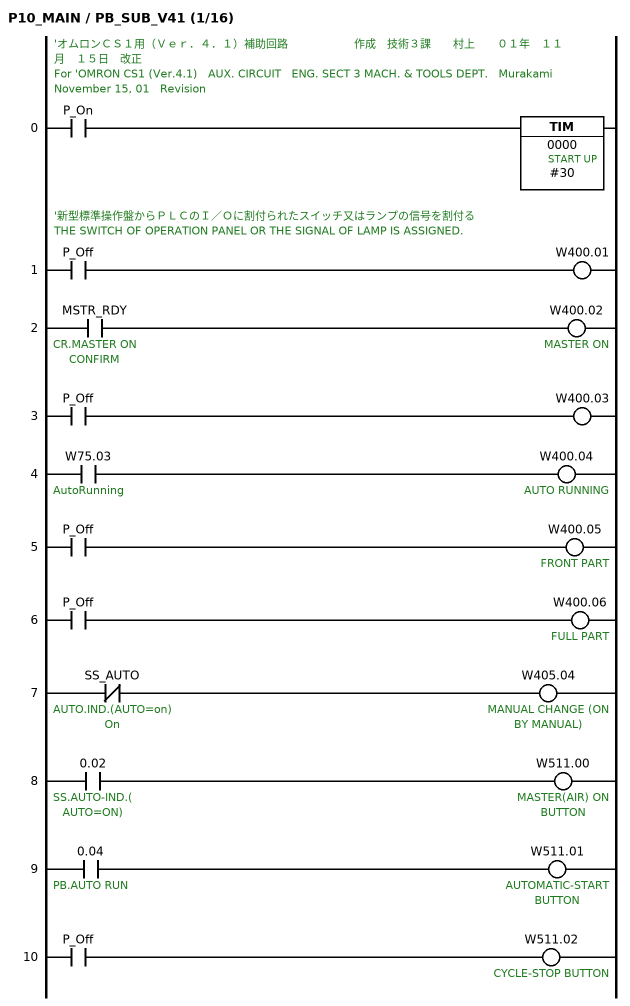
; [picture p72: P10_MAIN / PB_SUB_V41, rungs 0-10]
; rung 0: 'オムロンＣＳ１用（Ｖｅｒ．４．１）補助回路　　　　　　作成　技術３課　　村上　　０１年　１１月　１５日　改正 / For 'OMRON CS1 (Ver.4.1)   AUX. CIRCUIT   ENG. SECT 3 MACH. & TOOLS DEPT.   Murakami   November 15, 01   Revision
LD P_On
TIM 0000 #30  ; START UP
; rung 1: '新型標準操作盤からＰＬＣのＩ／Ｏに割付られたスイッチ又はランプの信号を割付る / THE SWITCH OF OPERATION PANEL OR THE SIGNAL OF LAMP IS ASSIGNED.
LD P_Off
OUT W400.01
; rung 2
LD MSTR_RDY  ; CR.MASTER ON CONFIRM
OUT W400.02  ; MASTER ON
; rung 3
LD P_Off
OUT W400.03
; rung 4
LD W75.03  ; AutoRunning
OUT W400.04  ; AUTO RUNNING
; rung 5
LD P_Off
OUT W400.05  ; FRONT PART
; rung 6
LD P_Off
OUT W400.06  ; FULL PART
; rung 7
LDNOT SS_AUTO  ; AUTO.IND.(AUTO=on) On
OUT W405.04  ; MANUAL CHANGE (ON BY MANUAL)
; rung 8
LD 0.02  ; SS.AUTO-IND.(AUTO=ON)
OUT W511.00  ; MASTER(AIR) ON BUTTON
; rung 9
LD 0.04  ; PB.AUTO RUN
OUT W511.01  ; AUTOMATIC-START BUTTON
; rung 10
LD P_Off
OUT W511.02  ; CYCLE-STOP BUTTON

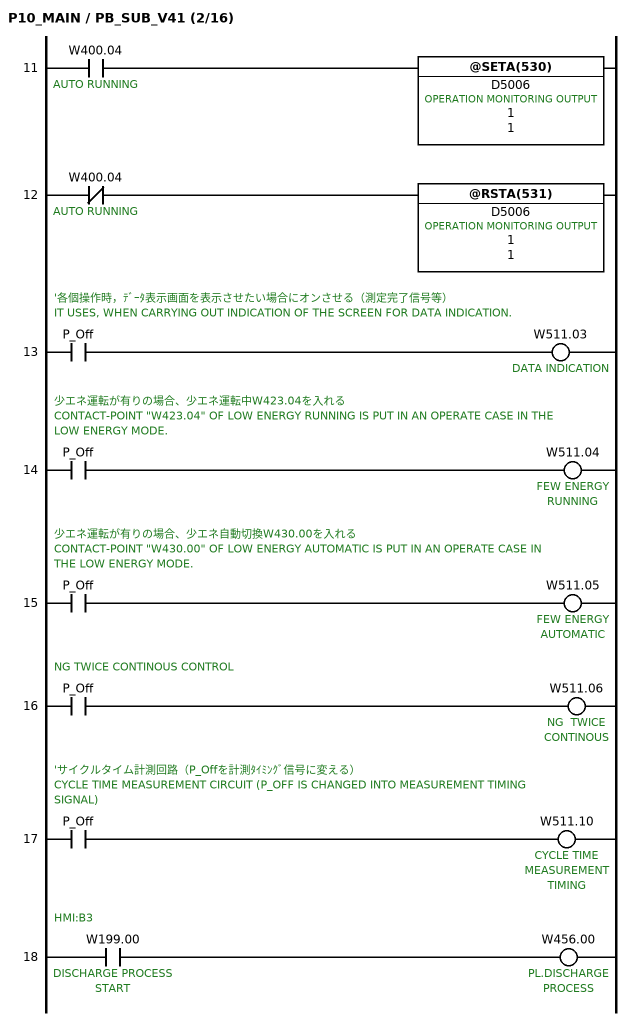
; rung 11
LD W400.04  ; AUTO RUNNING
@SETA(530) D5006 1 1  ; OPERATION MONITORING OUTPUT
; rung 12
LDNOT W400.04  ; AUTO RUNNING
@RSTA(531) D5006 1 1  ; OPERATION MONITORING OUTPUT
; rung 13: '各個操作時，ﾃﾞｰﾀ表示画面を表示させたい場合にオンさせる（測定完了信号等） / IT USES, WHEN CARRYING OUT INDICATION OF THE SCREEN FOR DATA INDICATION.
LD P_Off
OUT W511.03  ; DATA INDICATION
; rung 14: 少エネ運転が有りの場合、少エネ運転中W423.04を入れる / CONTACT-POINT "W423.04" OF LOW ENERGY RUNNING IS PUT IN AN OPERATE CASE IN THE LOW ENERGY MODE.
LD P_Off
OUT W511.04  ; FEW ENERGY RUNNING
; rung 15: 少エネ運転が有りの場合、少エネ自動切換W430.00を入れる / CONTACT-POINT "W430.00" OF LOW ENERGY AUTOMATIC IS PUT IN AN OPERATE CASE IN THE LOW ENERGY MODE.
LD P_Off
OUT W511.05  ; FEW ENERGY AUTOMATIC
; rung 16: NG TWICE CONTINOUS CONTROL
LD P_Off
OUT W511.06  ; NG  TWICE CONTINOUS
; rung 17: 'サイクルタイム計測回路（P_Offを計測ﾀｲﾐﾝｸﾞ信号に変える） / CYCLE TIME MEASUREMENT CIRCUIT (P_OFF IS CHANGED INTO MEASUREMENT TIMING SIGNAL)
LD P_Off
OUT W511.10  ; CYCLE TIME MEASUREMENT TIMING
; rung 18: HMI:B3
LD W199.00  ; DISCHARGE PROCESS START
OUT W456.00  ; PL.DISCHARGE PROCESS

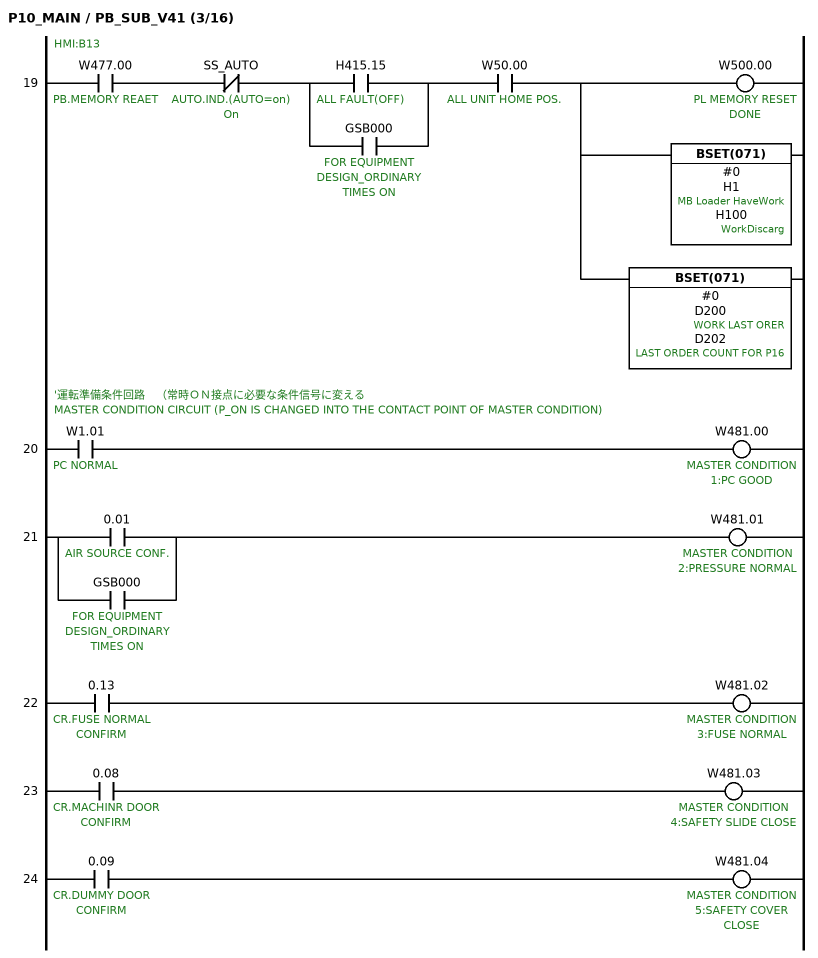
; rung 19: HMI:B13
LD W477.00  ; PB.MEMORY REAET
ANDNOT SS_AUTO  ; AUTO.IND.(AUTO=on) On
LD H415.15  ; ALL FAULT(OFF)
OR GSB000  ; FOR EQUIPMENT DESIGN_ORDINARY TIMES ON
ANDLD
AND W50.00  ; ALL UNIT HOME POS.
OUT W500.00  ; PL MEMORY RESET DONE
BSET(071) #0 H1 H100  ; MB Loader HaveWork, WorkDiscarg
BSET(071) #0 D200 D202  ; WORK LAST ORER, LAST ORDER COUNT FOR P16
; rung 20: '運転準備条件回路　（常時ＯＮ接点に必要な条件信号に変える / MASTER CONDITION CIRCUIT (P_ON IS CHANGED INTO THE CONTACT POINT OF MASTER CONDITION)
LD W1.01  ; PC NORMAL
OUT W481.00  ; MASTER CONDITION 1:PC GOOD
; rung 21
LD 0.01  ; AIR SOURCE CONF.
OR GSB000  ; FOR EQUIPMENT DESIGN_ORDINARY TIMES ON
OUT W481.01  ; MASTER CONDITION 2:PRESSURE NORMAL
; rung 22
LD 0.13  ; CR.FUSE NORMAL CONFIRM
OUT W481.02  ; MASTER CONDITION 3:FUSE NORMAL
; rung 23
LD 0.08  ; CR.MACHINR DOOR CONFIRM
OUT W481.03  ; MASTER CONDITION 4:SAFETY SLIDE CLOSE
; rung 24
LD 0.09  ; CR.DUMMY DOOR CONFIRM
OUT W481.04  ; MASTER CONDITION 5:SAFETY COVER CLOSE

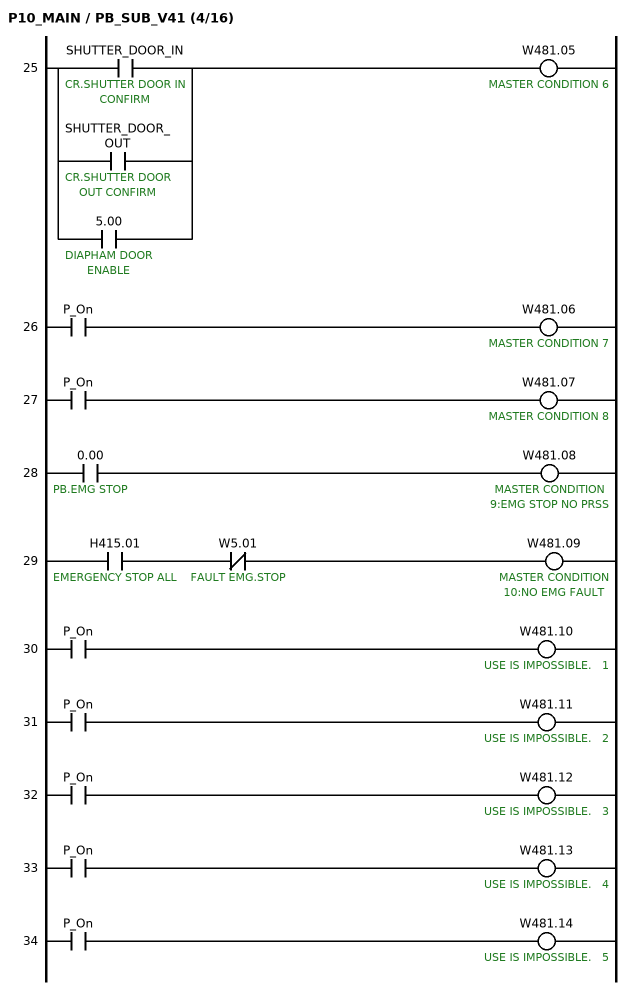
; rung 25
LD SHUTTER_DOOR_IN  ; CR.SHUTTER DOOR IN CONFIRM
OR SHUTTER_DOOR_OUT  ; CR.SHUTTER DOOR OUT CONFIRM
OR 5.00  ; DIAPHAM DOOR ENABLE
OUT W481.05  ; MASTER CONDITION 6
; rung 26
LD P_On
OUT W481.06  ; MASTER CONDITION 7
; rung 27
LD P_On
OUT W481.07  ; MASTER CONDITION 8
; rung 28
LD 0.00  ; PB.EMG STOP
OUT W481.08  ; MASTER CONDITION 9:EMG STOP NO PRSS
; rung 29
LD H415.01  ; EMERGENCY STOP ALL
ANDNOT W5.01  ; FAULT EMG.STOP
OUT W481.09  ; MASTER CONDITION 10:NO EMG FAULT
; rung 30
LD P_On
OUT W481.10  ; USE IS IMPOSSIBLE.   1
; rung 31
LD P_On
OUT W481.11  ; USE IS IMPOSSIBLE.   2
; rung 32
LD P_On
OUT W481.12  ; USE IS IMPOSSIBLE.   3
; rung 33
LD P_On
OUT W481.13  ; USE IS IMPOSSIBLE.   4
; rung 34
LD P_On
OUT W481.14  ; USE IS IMPOSSIBLE.   5

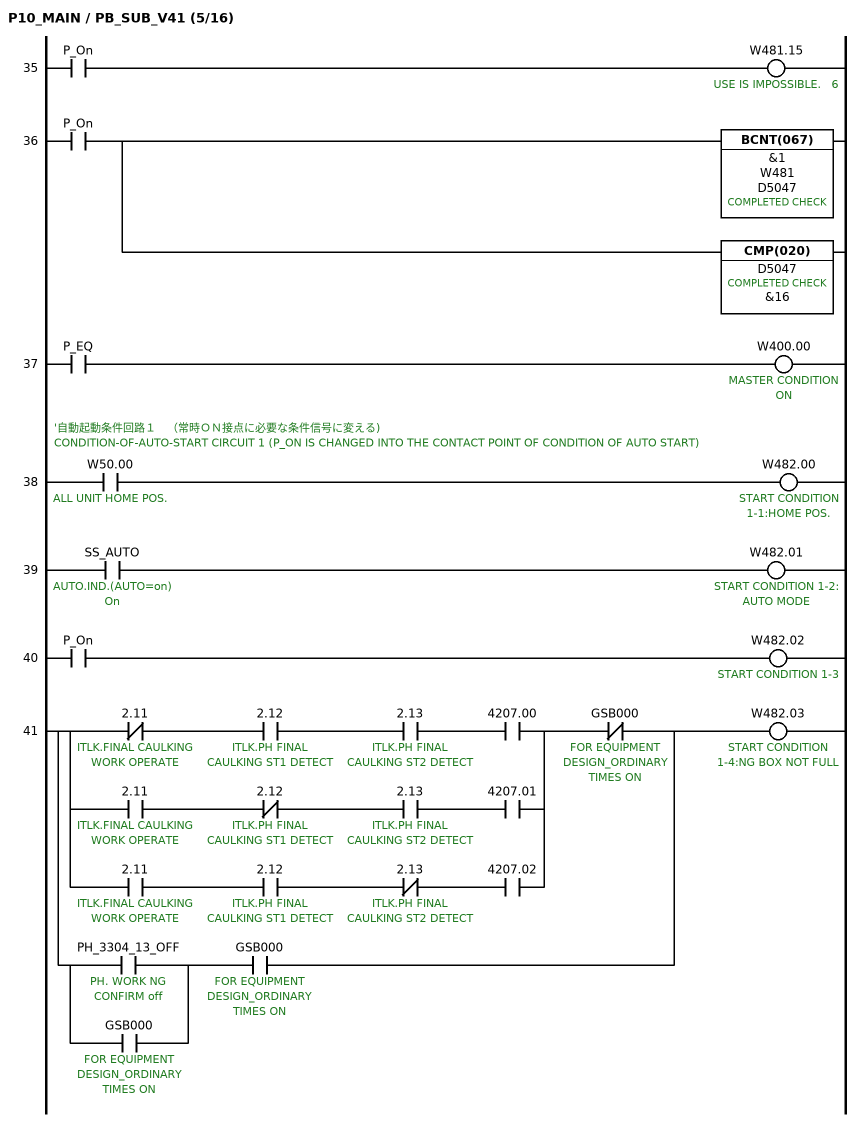
; rung 35
LD P_On
OUT W481.15  ; USE IS IMPOSSIBLE.   6
; rung 36
LD P_On
BCNT(067) &1 W481 D5047  ; COMPLETED CHECK
CMP(020) D5047 &16  ; COMPLETED CHECK
; rung 37
LD P_EQ
OUT W400.00  ; MASTER CONDITION ON
; rung 38: '自動起動条件回路１　（常時ＯＮ接点に必要な条件信号に変える) / CONDITION-OF-AUTO-START CIRCUIT 1 (P_ON IS CHANGED INTO THE CONTACT POINT OF CONDITION OF AUTO START)
LD W50.00  ; ALL UNIT HOME POS.
OUT W482.00  ; START CONDITION 1-1:HOME POS.
; rung 39
LD SS_AUTO  ; AUTO.IND.(AUTO=on) On
OUT W482.01  ; START CONDITION 1-2: AUTO MODE
; rung 40
LD P_On
OUT W482.02  ; START CONDITION 1-3
; rung 41
LDNOT 2.11  ; ITLK.FINAL CAULKING WORK OPERATE
AND 2.12  ; ITLK.PH FINAL CAULKING ST1 DETECT
AND 2.13  ; ITLK.PH FINAL CAULKING ST2 DETECT
AND 4207.00
LD 2.11  ; ITLK.FINAL CAULKING WORK OPERATE
ANDNOT 2.12  ; ITLK.PH FINAL CAULKING ST1 DETECT
AND 2.13  ; ITLK.PH FINAL CAULKING ST2 DETECT
AND 4207.01
ORLD
LD 2.11  ; ITLK.FINAL CAULKING WORK OPERATE
AND 2.12  ; ITLK.PH FINAL CAULKING ST1 DETECT
ANDNOT 2.13  ; ITLK.PH FINAL CAULKING ST2 DETECT
AND 4207.02
ORLD
ANDNOT GSB000  ; FOR EQUIPMENT DESIGN_ORDINARY TIMES ON
LD PH_3304_13_OFF  ; PH. WORK NG CONFIRM off
OR GSB000  ; FOR EQUIPMENT DESIGN_ORDINARY TIMES ON
AND GSB000  ; FOR EQUIPMENT DESIGN_ORDINARY TIMES ON
ORLD
OUT W482.03  ; START CONDITION 1-4:NG BOX NOT FULL

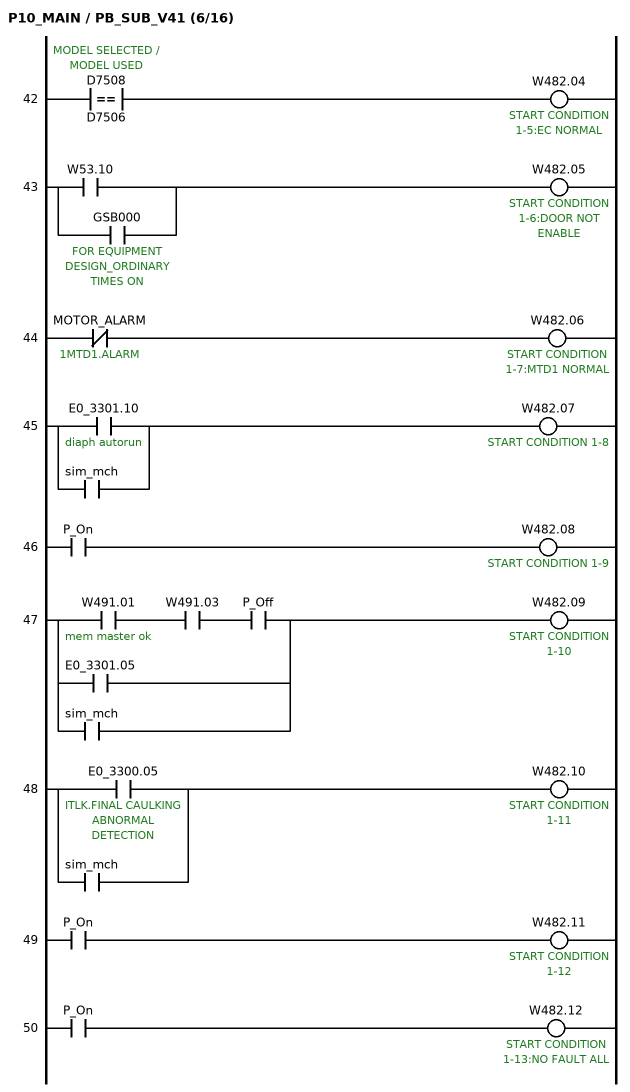
; rung 42
LD=(300) D7508 D7506  ; MODEL SELECTED, MODEL USED
OUT W482.04  ; START CONDITION 1-5:EC NORMAL
; rung 43
LD W53.10
OR GSB000  ; FOR EQUIPMENT DESIGN_ORDINARY TIMES ON
OUT W482.05  ; START CONDITION 1-6:DOOR NOT ENABLE
; rung 44
LDNOT MOTOR_ALARM  ; 1MTD1.ALARM
OUT W482.06  ; START CONDITION 1-7:MTD1 NORMAL
; rung 45
LD E0_3301.10  ; diaph autorun
OR sim_mch
OUT W482.07  ; START CONDITION 1-8
; rung 46
LD P_On
OUT W482.08  ; START CONDITION 1-9
; rung 47
LD W491.01  ; mem master ok
AND W491.03
AND P_Off
OR E0_3301.05
OR sim_mch
OUT W482.09  ; START CONDITION 1-10
; rung 48
LD E0_3300.05  ; ITLK.FINAL CAULKING ABNORMAL DETECTION
OR sim_mch
OUT W482.10  ; START CONDITION 1-11
; rung 49
LD P_On
OUT W482.11  ; START CONDITION 1-12
; rung 50
LD P_On
OUT W482.12  ; START CONDITION 1-13:NO FAULT ALL

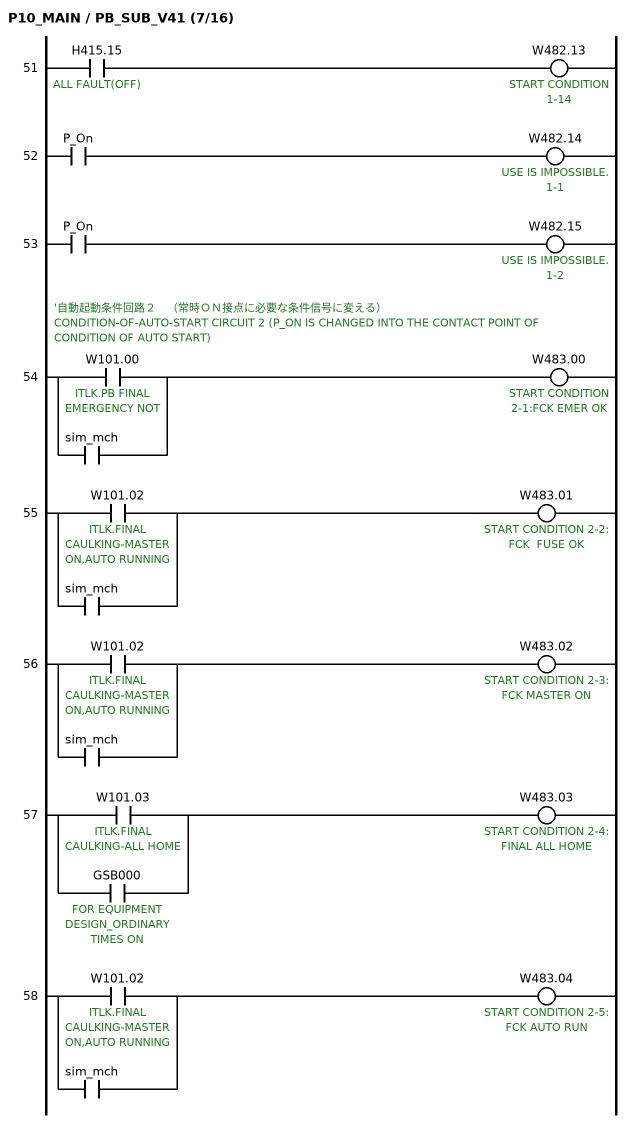
; rung 51
LD H415.15  ; ALL FAULT(OFF)
OUT W482.13  ; START CONDITION 1-14
; rung 52
LD P_On
OUT W482.14  ; USE IS IMPOSSIBLE.   1-1
; rung 53
LD P_On
OUT W482.15  ; USE IS IMPOSSIBLE.   1-2
; rung 54: '自動起動条件回路２　（常時ＯＮ接点に必要な条件信号に変える） / CONDITION-OF-AUTO-START CIRCUIT 2 (P_ON IS CHANGED INTO THE CONTACT POINT OF CONDITION OF AUTO START)
LD W101.00  ; ITLK.PB FINAL EMERGENCY NOT
OR sim_mch
OUT W483.00  ; START CONDITION 2-1:FCK EMER OK
; rung 55
LD W101.02  ; ITLK.FINAL CAULKING-MASTER ON,AUTO RUNNING
OR sim_mch
OUT W483.01  ; START CONDITION 2-2: FCK  FUSE OK
; rung 56
LD W101.02  ; ITLK.FINAL CAULKING-MASTER ON,AUTO RUNNING
OR sim_mch
OUT W483.02  ; START CONDITION 2-3: FCK MASTER ON
; rung 57
LD W101.03  ; ITLK.FINAL CAULKING-ALL HOME
OR GSB000  ; FOR EQUIPMENT DESIGN_ORDINARY TIMES ON
OUT W483.03  ; START CONDITION 2-4: FINAL ALL HOME
; rung 58
LD W101.02  ; ITLK.FINAL CAULKING-MASTER ON,AUTO RUNNING
OR sim_mch
OUT W483.04  ; START CONDITION 2-5: FCK AUTO RUN

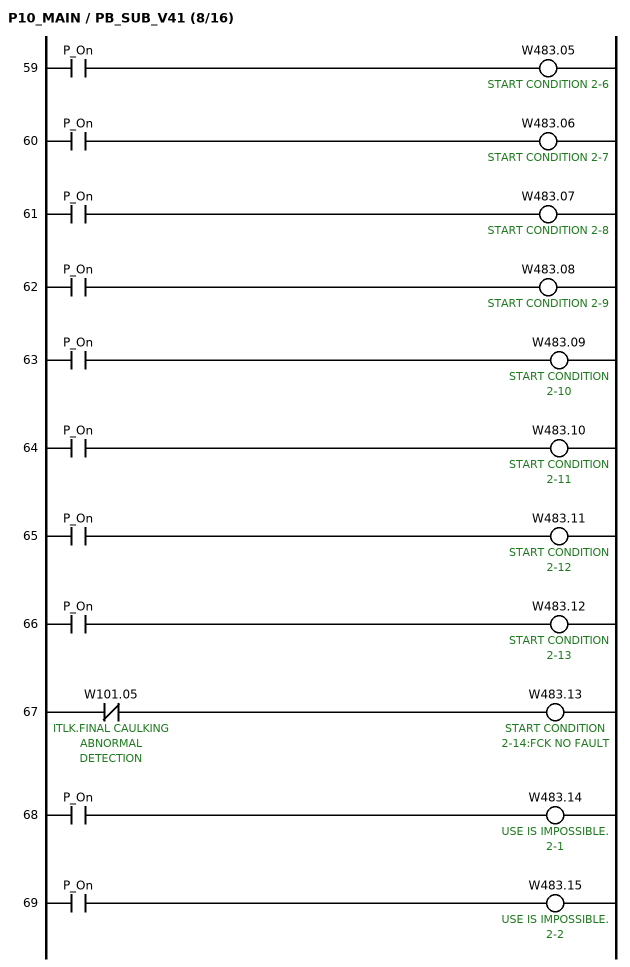
; rung 59
LD P_On
OUT W483.05  ; START CONDITION 2-6
; rung 60
LD P_On
OUT W483.06  ; START CONDITION 2-7
; rung 61
LD P_On
OUT W483.07  ; START CONDITION 2-8
; rung 62
LD P_On
OUT W483.08  ; START CONDITION 2-9
; rung 63
LD P_On
OUT W483.09  ; START CONDITION 2-10
; rung 64
LD P_On
OUT W483.10  ; START CONDITION 2-11
; rung 65
LD P_On
OUT W483.11  ; START CONDITION 2-12
; rung 66
LD P_On
OUT W483.12  ; START CONDITION 2-13
; rung 67
LDNOT W101.05  ; ITLK.FINAL CAULKING ABNORMAL DETECTION
OUT W483.13  ; START CONDITION 2-14:FCK NO FAULT
; rung 68
LD P_On
OUT W483.14  ; USE IS IMPOSSIBLE.   2-1
; rung 69
LD P_On
OUT W483.15  ; USE IS IMPOSSIBLE.   2-2

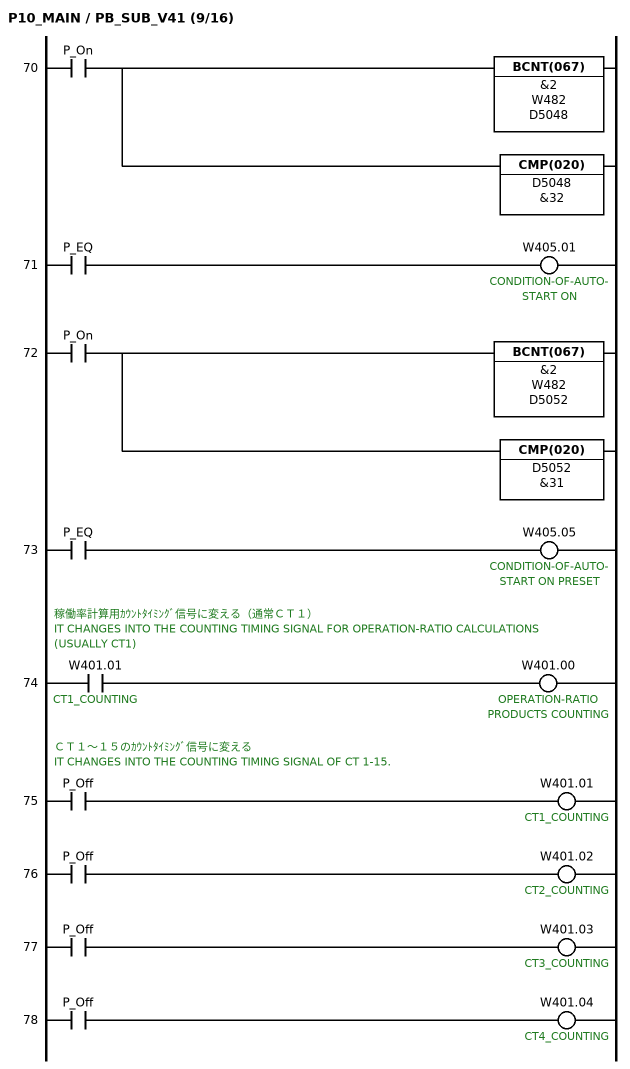
; rung 70
LD P_On
BCNT(067) &2 W482 D5048
CMP(020) D5048 &32
; rung 71
LD P_EQ
OUT W405.01  ; CONDITION-OF-AUTO-START ON
; rung 72
LD P_On
BCNT(067) &2 W482 D5052
CMP(020) D5052 &31
; rung 73
LD P_EQ
OUT W405.05  ; CONDITION-OF-AUTO-START ON PRESET
; rung 74: 稼働率計算用ｶｳﾝﾄﾀｲﾐﾝｸﾞ信号に変える（通常ＣＴ１） / IT CHANGES INTO THE COUNTING TIMING SIGNAL FOR OPERATION-RATIO CALCULATIONS (USUALLY CT1)
LD W401.01  ; CT1_COUNTING
OUT W401.00  ; OPERATION-RATIO PRODUCTS COUNTING
; rung 75: ＣＴ１～１５のｶｳﾝﾄﾀｲﾐﾝｸﾞ信号に変える / IT CHANGES INTO THE COUNTING TIMING SIGNAL OF CT 1-15.
LD P_Off
OUT W401.01  ; CT1_COUNTING
; rung 76
LD P_Off
OUT W401.02  ; CT2_COUNTING
; rung 77
LD P_Off
OUT W401.03  ; CT3_COUNTING
; rung 78
LD P_Off
OUT W401.04  ; CT4_COUNTING

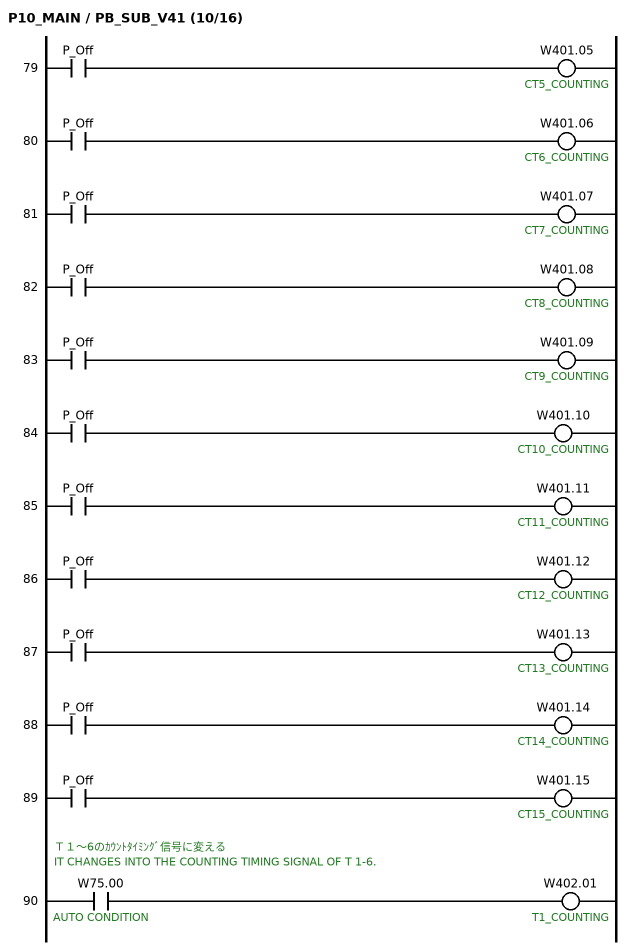
; rung 79
LD P_Off
OUT W401.05  ; CT5_COUNTING
; rung 80
LD P_Off
OUT W401.06  ; CT6_COUNTING
; rung 81
LD P_Off
OUT W401.07  ; CT7_COUNTING
; rung 82
LD P_Off
OUT W401.08  ; CT8_COUNTING
; rung 83
LD P_Off
OUT W401.09  ; CT9_COUNTING
; rung 84
LD P_Off
OUT W401.10  ; CT10_COUNTING
; rung 85
LD P_Off
OUT W401.11  ; CT11_COUNTING
; rung 86
LD P_Off
OUT W401.12  ; CT12_COUNTING
; rung 87
LD P_Off
OUT W401.13  ; CT13_COUNTING
; rung 88
LD P_Off
OUT W401.14  ; CT14_COUNTING
; rung 89
LD P_Off
OUT W401.15  ; CT15_COUNTING
; rung 90: Ｔ１～6のｶｳﾝﾄﾀｲﾐﾝｸﾞ信号に変える / IT CHANGES INTO THE COUNTING TIMING SIGNAL OF T 1-6.
LD W75.00  ; AUTO CONDITION
OUT W402.01  ; T1_COUNTING

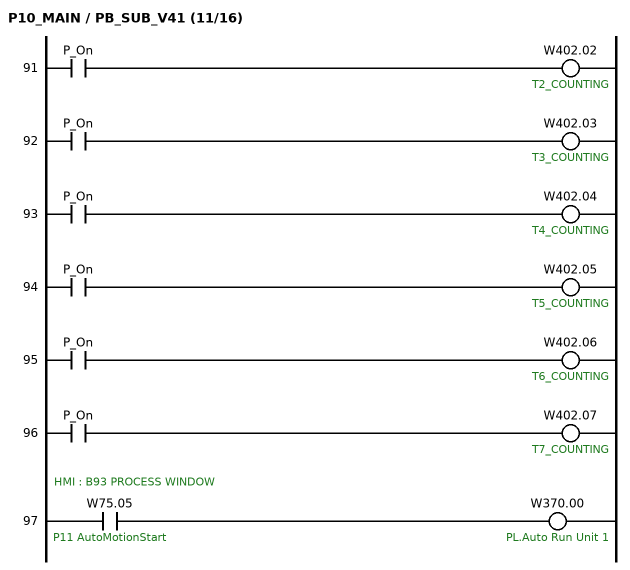
; rung 91
LD P_On
OUT W402.02  ; T2_COUNTING
; rung 92
LD P_On
OUT W402.03  ; T3_COUNTING
; rung 93
LD P_On
OUT W402.04  ; T4_COUNTING
; rung 94
LD P_On
OUT W402.05  ; T5_COUNTING
; rung 95
LD P_On
OUT W402.06  ; T6_COUNTING
; rung 96
LD P_On
OUT W402.07  ; T7_COUNTING
; rung 97: HMI : B93 PROCESS WINDOW
LD W75.05  ; P11 AutoMotionStart
OUT W370.00  ; PL.Auto Run Unit 1

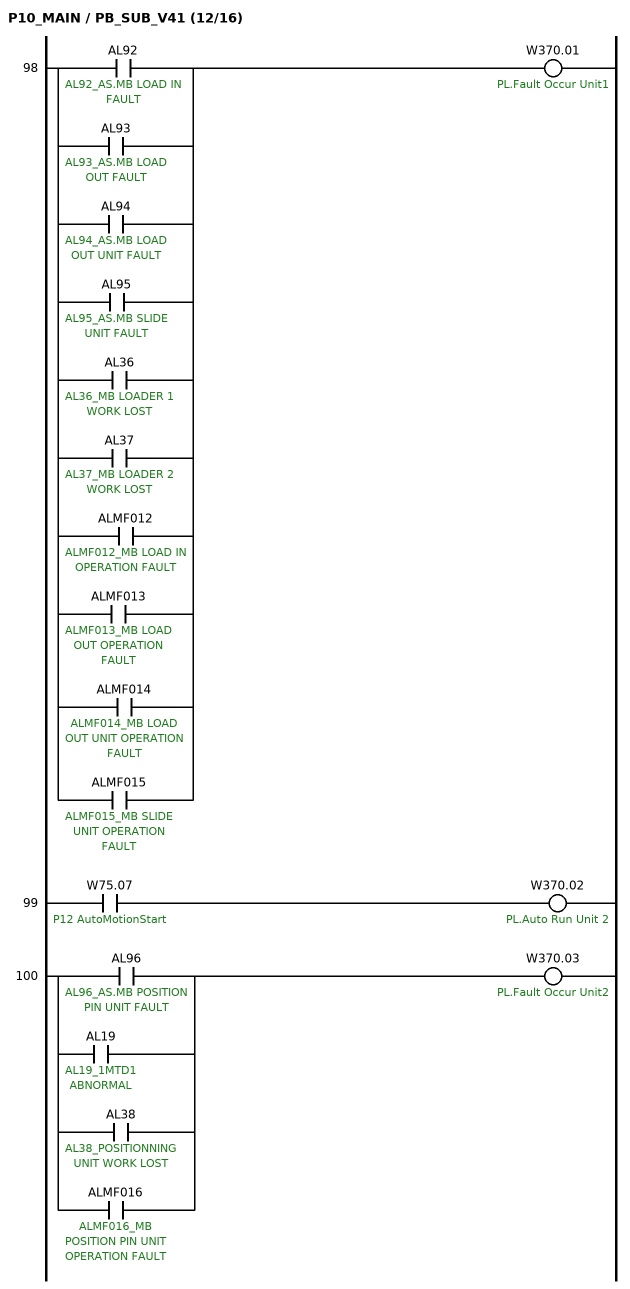
; rung 98
LD AL92  ; AL92_AS.MB LOAD IN FAULT
OR AL93  ; AL93_AS.MB LOAD OUT FAULT
OR AL94  ; AL94_AS.MB LOAD OUT UNIT FAULT
OR AL95  ; AL95_AS.MB SLIDE UNIT FAULT
OR AL36  ; AL36_MB LOADER 1 WORK LOST
OR AL37  ; AL37_MB LOADER 2 WORK LOST
OR ALMF012  ; ALMF012_MB LOAD IN OPERATION FAULT
OR ALMF013  ; ALMF013_MB LOAD OUT OPERATION FAULT
OR ALMF014  ; ALMF014_MB LOAD OUT UNIT OPERATION FAULT
OR ALMF015  ; ALMF015_MB SLIDE UNIT OPERATION FAULT
OUT W370.01  ; PL.Fault Occur Unit1
; rung 99
LD W75.07  ; P12 AutoMotionStart
OUT W370.02  ; PL.Auto Run Unit 2
; rung 100
LD AL96  ; AL96_AS.MB POSITION PIN UNIT FAULT
OR AL19  ; AL19_1MTD1 ABNORMAL
OR AL38  ; AL38_POSITIONNING UNIT WORK LOST
OR ALMF016  ; ALMF016_MB POSITION PIN UNIT OPERATION FAULT
OUT W370.03  ; PL.Fault Occur Unit2

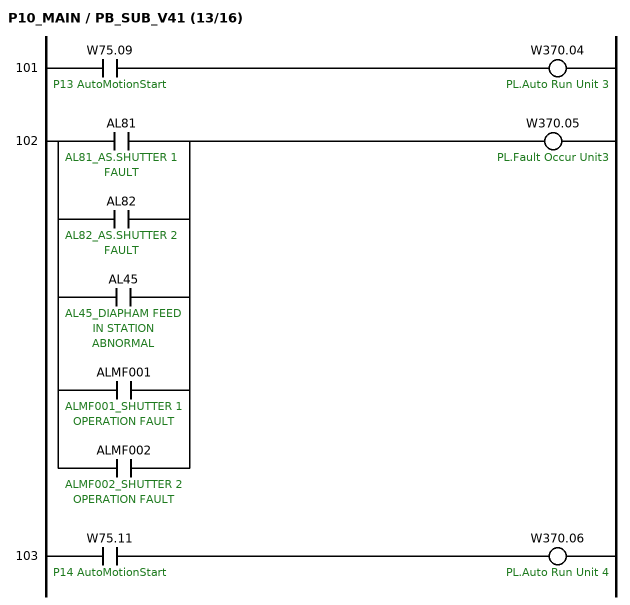
; rung 101
LD W75.09  ; P13 AutoMotionStart
OUT W370.04  ; PL.Auto Run Unit 3
; rung 102
LD AL81  ; AL81_AS.SHUTTER 1 FAULT
OR AL82  ; AL82_AS.SHUTTER 2 FAULT
OR AL45  ; AL45_DIAPHAM FEED IN STATION ABNORMAL
OR ALMF001  ; ALMF001_SHUTTER 1 OPERATION FAULT
OR ALMF002  ; ALMF002_SHUTTER 2 OPERATION FAULT
OUT W370.05  ; PL.Fault Occur Unit3
; rung 103
LD W75.11  ; P14 AutoMotionStart
OUT W370.06  ; PL.Auto Run Unit 4

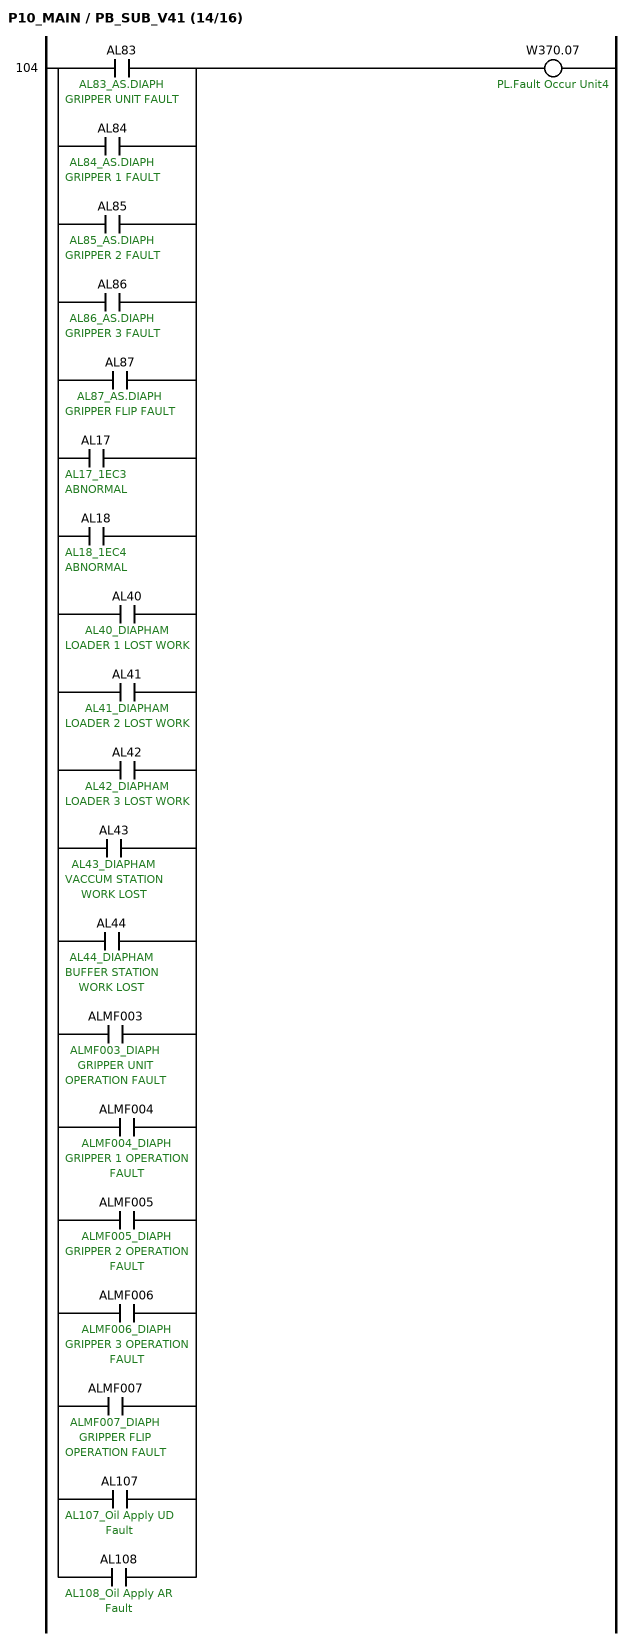
; rung 104
LD AL83  ; AL83_AS.DIAPH GRIPPER UNIT FAULT
OR AL84  ; AL84_AS.DIAPH GRIPPER 1 FAULT
OR AL85  ; AL85_AS.DIAPH GRIPPER 2 FAULT
OR AL86  ; AL86_AS.DIAPH GRIPPER 3 FAULT
OR AL87  ; AL87_AS.DIAPH GRIPPER FLIP FAULT
OR AL17  ; AL17_1EC3 ABNORMAL
OR AL18  ; AL18_1EC4 ABNORMAL
OR AL40  ; AL40_DIAPHAM LOADER 1 LOST WORK
OR AL41  ; AL41_DIAPHAM LOADER 2 LOST WORK
OR AL42  ; AL42_DIAPHAM LOADER 3 LOST WORK
OR AL43  ; AL43_DIAPHAM VACCUM STATION WORK LOST
OR AL44  ; AL44_DIAPHAM BUFFER STATION WORK LOST
OR ALMF003  ; ALMF003_DIAPH GRIPPER UNIT OPERATION FAULT
OR ALMF004  ; ALMF004_DIAPH GRIPPER 1 OPERATION FAULT
OR ALMF005  ; ALMF005_DIAPH GRIPPER 2 OPERATION FAULT
OR ALMF006  ; ALMF006_DIAPH GRIPPER 3 OPERATION FAULT
OR ALMF007  ; ALMF007_DIAPH GRIPPER FLIP OPERATION FAULT
OR AL107  ; AL107_Oil Apply UD Fault
OR AL108  ; AL108_Oil Apply AR Fault
OUT W370.07  ; PL.Fault Occur Unit4

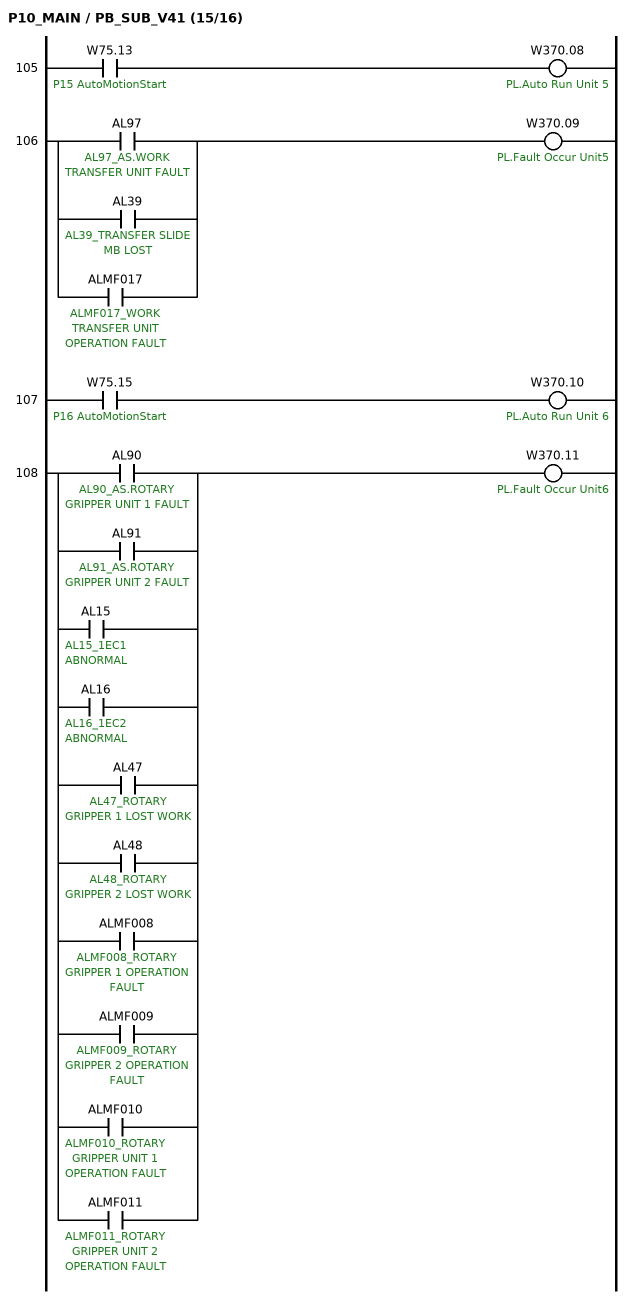
; rung 105
LD W75.13  ; P15 AutoMotionStart
OUT W370.08  ; PL.Auto Run Unit 5
; rung 106
LD AL97  ; AL97_AS.WORK TRANSFER UNIT FAULT
OR AL39  ; AL39_TRANSFER SLIDE MB LOST
OR ALMF017  ; ALMF017_WORK TRANSFER UNIT OPERATION FAULT
OUT W370.09  ; PL.Fault Occur Unit5
; rung 107
LD W75.15  ; P16 AutoMotionStart
OUT W370.10  ; PL.Auto Run Unit 6
; rung 108
LD AL90  ; AL90_AS.ROTARY GRIPPER UNIT 1 FAULT
OR AL91  ; AL91_AS.ROTARY GRIPPER UNIT 2 FAULT
OR AL15  ; AL15_1EC1 ABNORMAL
OR AL16  ; AL16_1EC2 ABNORMAL
OR AL47  ; AL47_ROTARY GRIPPER 1 LOST WORK
OR AL48  ; AL48_ROTARY GRIPPER 2 LOST WORK
OR ALMF008  ; ALMF008_ROTARY GRIPPER 1 OPERATION FAULT
OR ALMF009  ; ALMF009_ROTARY GRIPPER 2 OPERATION FAULT
OR ALMF010  ; ALMF010_ROTARY GRIPPER UNIT 1 OPERATION FAULT
OR ALMF011  ; ALMF011_ROTARY GRIPPER UNIT 2 OPERATION FAULT
OUT W370.11  ; PL.Fault Occur Unit6

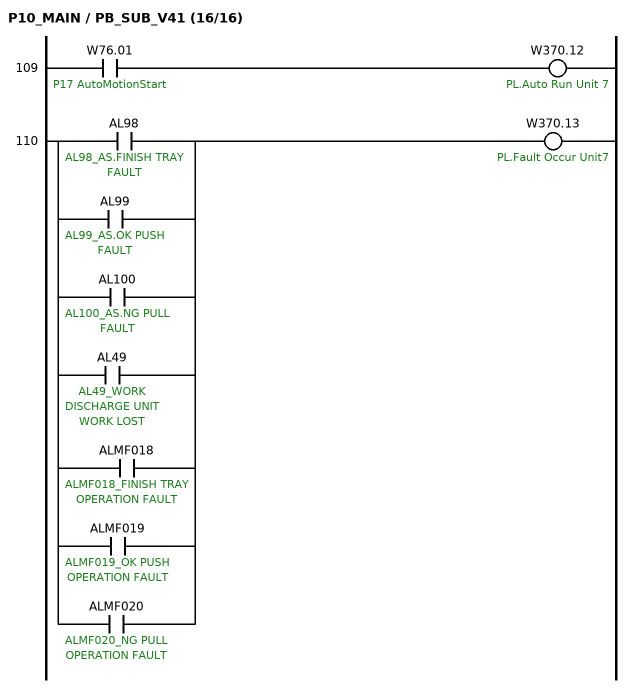
; rung 109
LD W76.01  ; P17 AutoMotionStart
OUT W370.12  ; PL.Auto Run Unit 7
; rung 110
LD AL98  ; AL98_AS.FINISH TRAY FAULT
OR AL99  ; AL99_AS.OK PUSH FAULT
OR AL100  ; AL100_AS.NG PULL FAULT
OR AL49  ; AL49_WORK DISCHARGE UNIT WORK LOST
OR ALMF018  ; ALMF018_FINISH TRAY OPERATION FAULT
OR ALMF019  ; ALMF019_OK PUSH OPERATION FAULT
OR ALMF020  ; ALMF020_NG PULL OPERATION FAULT
OUT W370.13  ; PL.Fault Occur Unit7

### Section PB_VTMAIN_V41

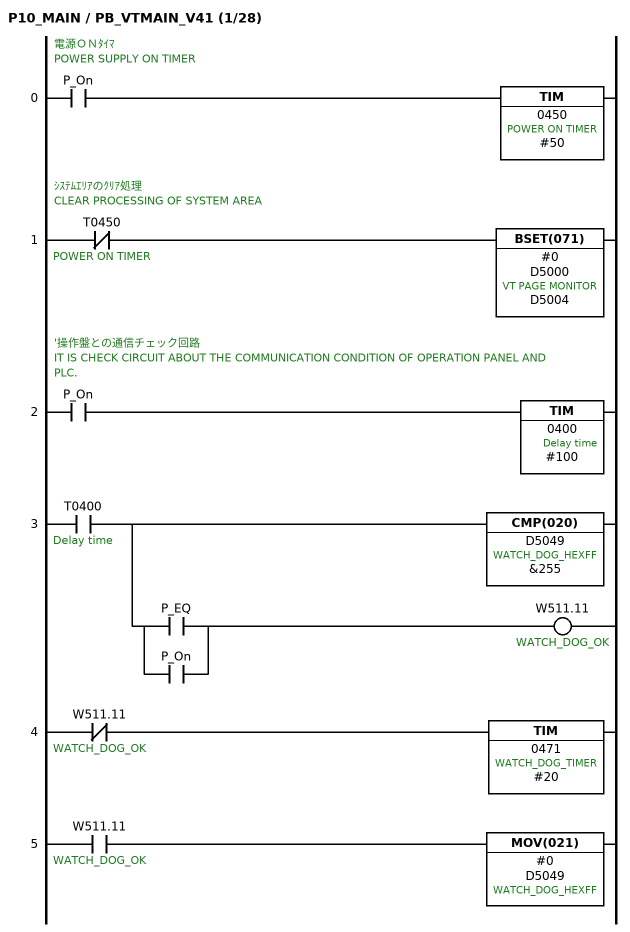
; rung 0: 電源ＯＮﾀｲﾏ / POWER SUPPLY ON TIMER
LD P_On
TIM 0450 #50  ; POWER ON TIMER
; rung 1: ｼｽﾃﾑｴﾘｱのｸﾘｱ処理 / CLEAR PROCESSING OF SYSTEM AREA
LDNOT T0450  ; POWER ON TIMER
BSET(071) #0 D5000 D5004  ; VT PAGE MONITOR
; rung 2: '操作盤との通信チェック回路 / IT IS CHECK CIRCUIT ABOUT THE COMMUNICATION CONDITION OF OPERATION PANEL AND PLC.
LD P_On
TIM 0400 #100  ; Delay time
; rung 3
LD T0400  ; Delay time
CMP(020) D5049 &255  ; WATCH_DOG_HEXFF
LD P_EQ
OR P_On
ANDLD
OUT W511.11  ; WATCH_DOG_OK
; rung 4
LDNOT W511.11  ; WATCH_DOG_OK
TIM 0471 #20  ; WATCH_DOG_TIMER
; rung 5
LD W511.11  ; WATCH_DOG_OK
MOV(021) #0 D5049  ; WATCH_DOG_HEXFF

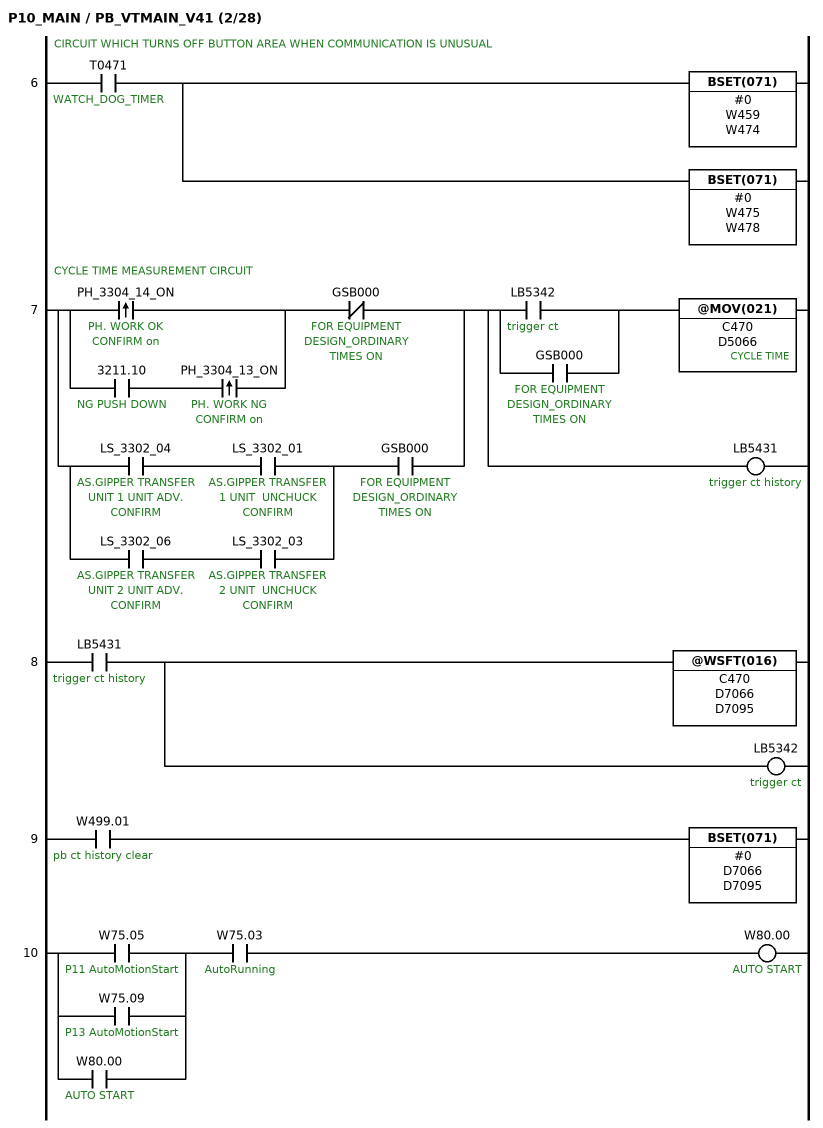
; rung 6: CIRCUIT WHICH TURNS OFF BUTTON AREA WHEN COMMUNICATION IS UNUSUAL
LD T0471  ; WATCH_DOG_TIMER
BSET(071) #0 W459 W474
BSET(071) #0 W475 W478
; rung 7: CYCLE TIME MEASUREMENT CIRCUIT
@LD PH_3304_14_ON  ; PH. WORK OK CONFIRM on
LD 3211.10  ; NG PUSH DOWN
@AND PH_3304_13_ON  ; PH. WORK NG CONFIRM on
ORLD
ANDNOT GSB000  ; FOR EQUIPMENT DESIGN_ORDINARY TIMES ON
LD LS_3302_04  ; AS.GIPPER TRANSFER UNIT 1 UNIT ADV. CONFIRM
AND LS_3302_01  ; AS.GIPPER TRANSFER 1 UNIT  UNCHUCK CONFIRM
LD LS_3302_06  ; AS.GIPPER TRANSFER UNIT 2 UNIT ADV. CONFIRM
AND LS_3302_03  ; AS.GIPPER TRANSFER 2 UNIT  UNCHUCK CONFIRM
ORLD
AND GSB000  ; FOR EQUIPMENT DESIGN_ORDINARY TIMES ON
ORLD
OUT TR0
LD LB5342  ; trigger ct
OR GSB000  ; FOR EQUIPMENT DESIGN_ORDINARY TIMES ON
ANDLD
@MOV(021) C470 D5066  ; CYCLE TIME
LD TR0
OUT LB5431  ; trigger ct history
; rung 8
LD LB5431  ; trigger ct history
@WSFT(016) C470 D7066 D7095
OUT LB5342  ; trigger ct
; rung 9
LD W499.01  ; pb ct history clear
BSET(071) #0 D7066 D7095
; rung 10
LD W75.05  ; P11 AutoMotionStart
OR W75.09  ; P13 AutoMotionStart
OR W80.00  ; AUTO START
AND W75.03  ; AutoRunning
OUT W80.00  ; AUTO START

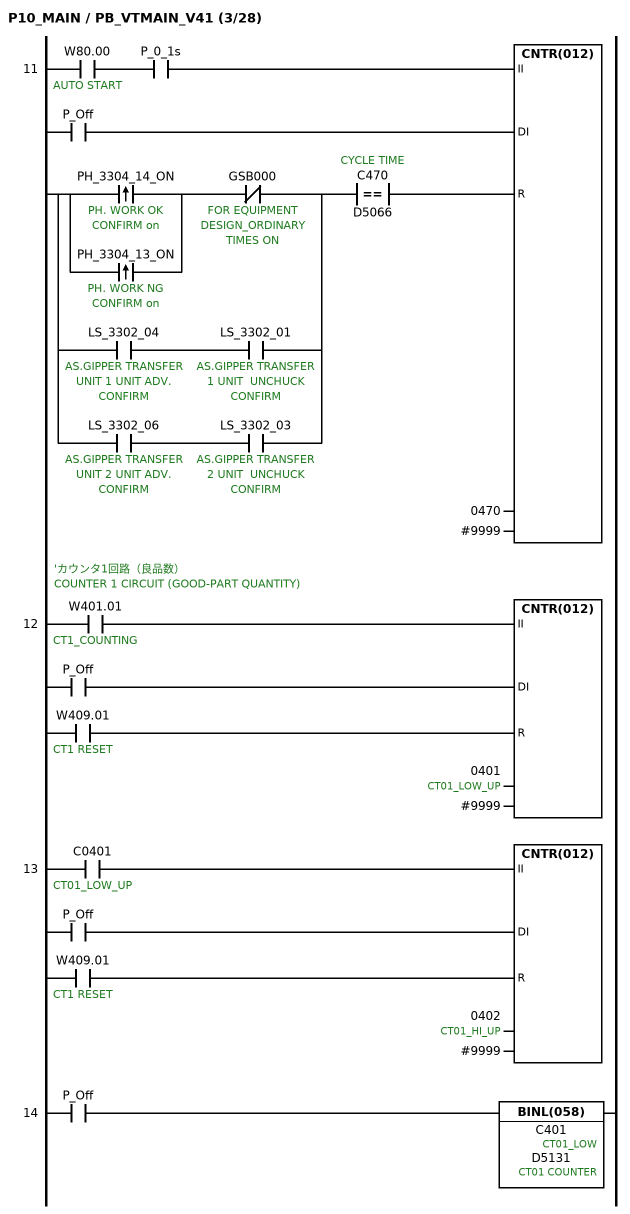
; rung 11
LD W80.00  ; AUTO START
AND P_0_1s
LD P_Off
@LD PH_3304_14_ON  ; PH. WORK OK CONFIRM on
@OR PH_3304_13_ON  ; PH. WORK NG CONFIRM on
ANDNOT GSB000  ; FOR EQUIPMENT DESIGN_ORDINARY TIMES ON
LD LS_3302_04  ; AS.GIPPER TRANSFER UNIT 1 UNIT ADV. CONFIRM
AND LS_3302_01  ; AS.GIPPER TRANSFER 1 UNIT  UNCHUCK CONFIRM
ORLD
LD LS_3302_06  ; AS.GIPPER TRANSFER UNIT 2 UNIT ADV. CONFIRM
AND LS_3302_03  ; AS.GIPPER TRANSFER 2 UNIT  UNCHUCK CONFIRM
ORLD
AND=(300) C470 D5066  ; CYCLE TIME
CNTR(012) 0470 #9999
; rung 12: 'カウンタ1回路（良品数） / COUNTER 1 CIRCUIT (GOOD-PART QUANTITY)
LD W401.01  ; CT1_COUNTING
LD P_Off
LD W409.01  ; CT1 RESET
CNTR(012) 0401 #9999  ; CT01_LOW_UP
; rung 13
LD C0401  ; CT01_LOW_UP
LD P_Off
LD W409.01  ; CT1 RESET
CNTR(012) 0402 #9999  ; CT01_HI_UP
; rung 14
LD P_Off
BINL(058) C401 D5131  ; CT01_LOW, CT01 COUNTER

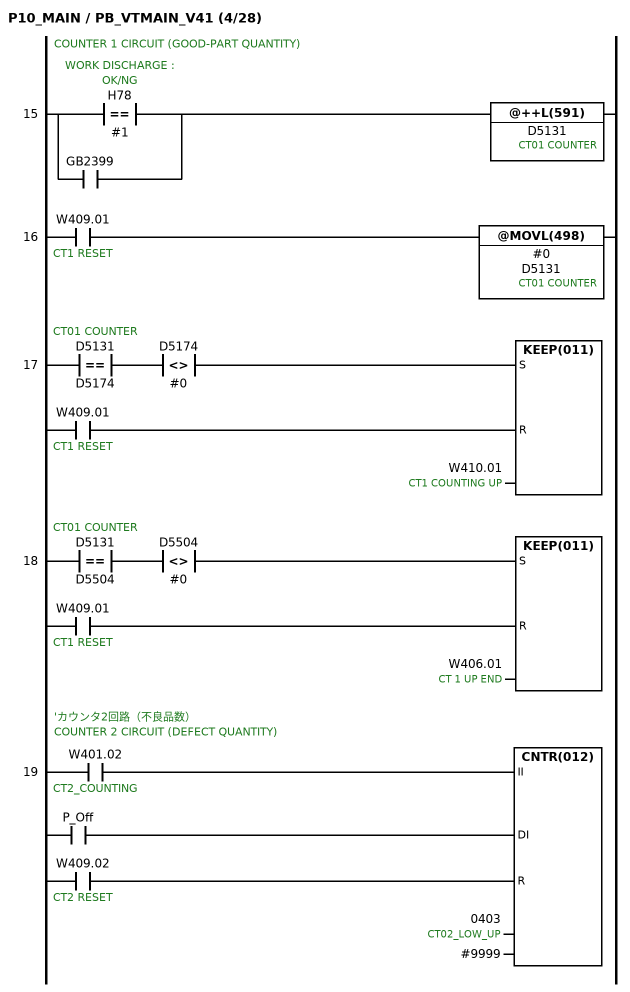
; rung 15: COUNTER 1 CIRCUIT (GOOD-PART QUANTITY)
LD=(300) H78 #1  ; WORK DISCHARGE : OK/NG
OR GB2399
@++L(591) D5131  ; CT01 COUNTER
; rung 16
LD W409.01  ; CT1 RESET
@MOVL(498) #0 D5131  ; CT01 COUNTER
; rung 17
LD=L(301) D5131 D5174  ; CT01 COUNTER
AND<>L(306) D5174 #0
LD W409.01  ; CT1 RESET
KEEP(011) W410.01  ; CT1 COUNTING UP
; rung 18
LD=L(301) D5131 D5504  ; CT01 COUNTER
AND<>L(306) D5504 #0
LD W409.01  ; CT1 RESET
KEEP(011) W406.01  ; CT 1 UP END
; rung 19: 'カウンタ2回路（不良品数） / COUNTER 2 CIRCUIT (DEFECT QUANTITY)
LD W401.02  ; CT2_COUNTING
LD P_Off
LD W409.02  ; CT2 RESET
CNTR(012) 0403 #9999  ; CT02_LOW_UP

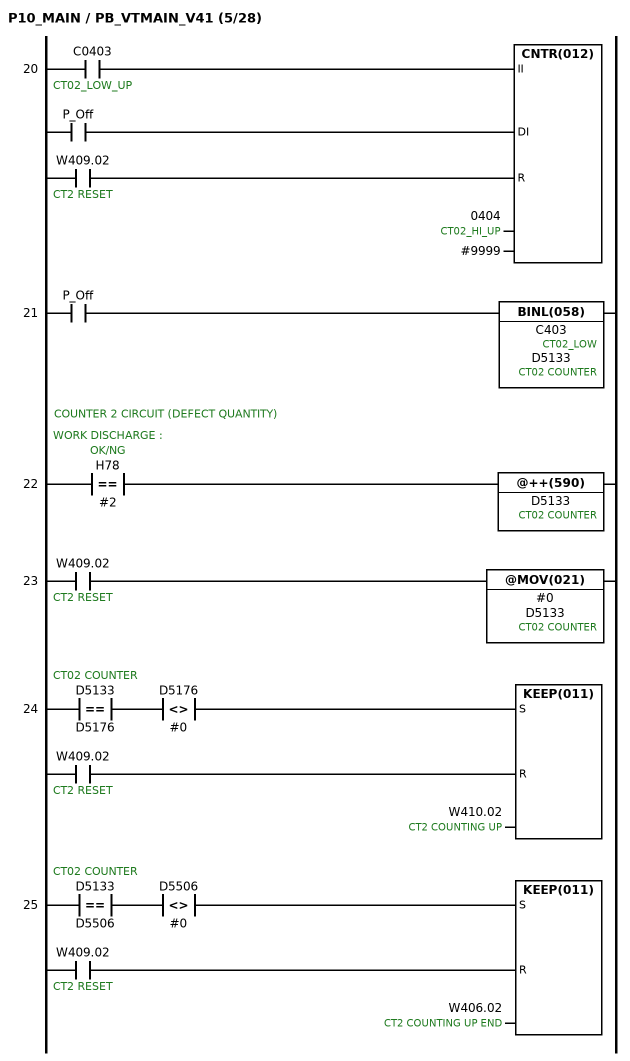
; rung 20
LD C0403  ; CT02_LOW_UP
LD P_Off
LD W409.02  ; CT2 RESET
CNTR(012) 0404 #9999  ; CT02_HI_UP
; rung 21
LD P_Off
BINL(058) C403 D5133  ; CT02_LOW, CT02 COUNTER
; rung 22: COUNTER 2 CIRCUIT (DEFECT QUANTITY)
LD=(300) H78 #2  ; WORK DISCHARGE : OK/NG
@++(590) D5133  ; CT02 COUNTER
; rung 23
LD W409.02  ; CT2 RESET
@MOV(021) #0 D5133  ; CT02 COUNTER
; rung 24
LD=L(301) D5133 D5176  ; CT02 COUNTER
AND<>L(306) D5176 #0
LD W409.02  ; CT2 RESET
KEEP(011) W410.02  ; CT2 COUNTING UP
; rung 25
LD=L(301) D5133 D5506  ; CT02 COUNTER
AND<>L(306) D5506 #0
LD W409.02  ; CT2 RESET
KEEP(011) W406.02  ; CT2 COUNTING UP END

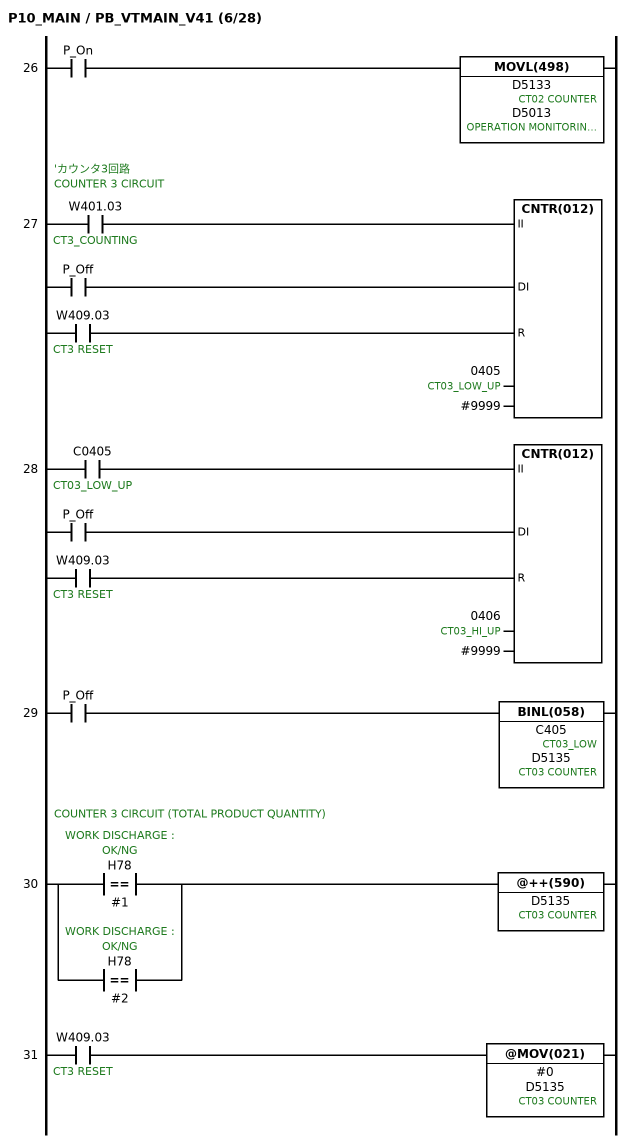
; rung 26
LD P_On
MOVL(498) D5133 D5013  ; CT02 COUNTER, OPERATION MONITORING TRANSMISSION
; rung 27: 'カウンタ3回路 / COUNTER 3 CIRCUIT
LD W401.03  ; CT3_COUNTING
LD P_Off
LD W409.03  ; CT3 RESET
CNTR(012) 0405 #9999  ; CT03_LOW_UP
; rung 28
LD C0405  ; CT03_LOW_UP
LD P_Off
LD W409.03  ; CT3 RESET
CNTR(012) 0406 #9999  ; CT03_HI_UP
; rung 29
LD P_Off
BINL(058) C405 D5135  ; CT03_LOW, CT03 COUNTER
; rung 30: COUNTER 3 CIRCUIT (TOTAL PRODUCT QUANTITY)
LD=(300) H78 #1  ; WORK DISCHARGE : OK/NG
OR=(300) H78 #2  ; WORK DISCHARGE : OK/NG
@++(590) D5135  ; CT03 COUNTER
; rung 31
LD W409.03  ; CT3 RESET
@MOV(021) #0 D5135  ; CT03 COUNTER

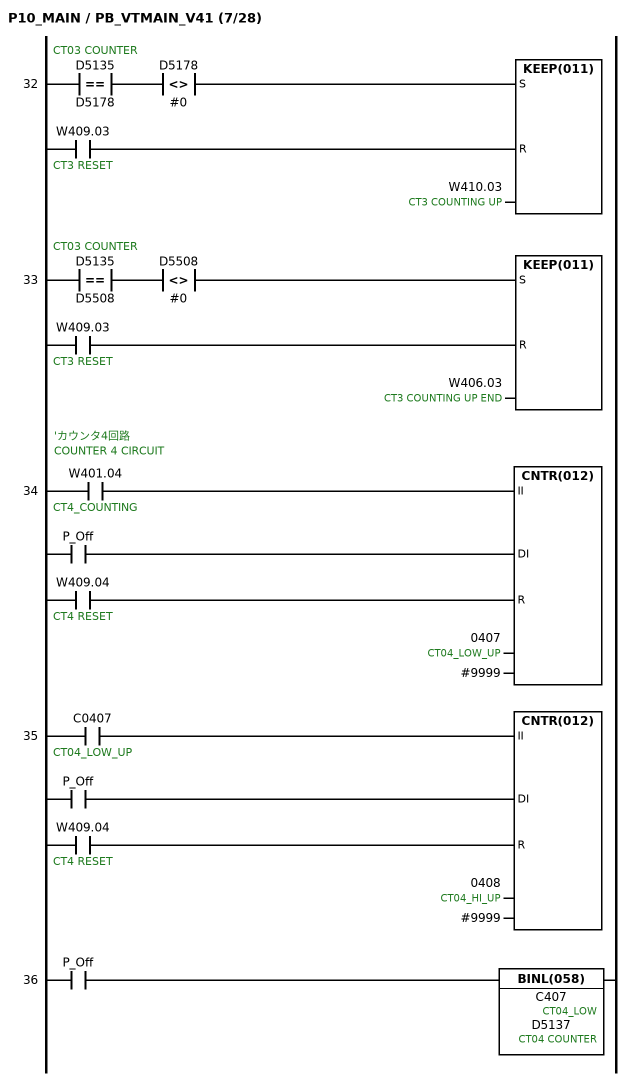
; rung 32
LD=L(301) D5135 D5178  ; CT03 COUNTER
AND<>L(306) D5178 #0
LD W409.03  ; CT3 RESET
KEEP(011) W410.03  ; CT3 COUNTING UP
; rung 33
LD=L(301) D5135 D5508  ; CT03 COUNTER
AND<>L(306) D5508 #0
LD W409.03  ; CT3 RESET
KEEP(011) W406.03  ; CT3 COUNTING UP END
; rung 34: 'カウンタ4回路 / COUNTER 4 CIRCUIT
LD W401.04  ; CT4_COUNTING
LD P_Off
LD W409.04  ; CT4 RESET
CNTR(012) 0407 #9999  ; CT04_LOW_UP
; rung 35
LD C0407  ; CT04_LOW_UP
LD P_Off
LD W409.04  ; CT4 RESET
CNTR(012) 0408 #9999  ; CT04_HI_UP
; rung 36
LD P_Off
BINL(058) C407 D5137  ; CT04_LOW, CT04 COUNTER

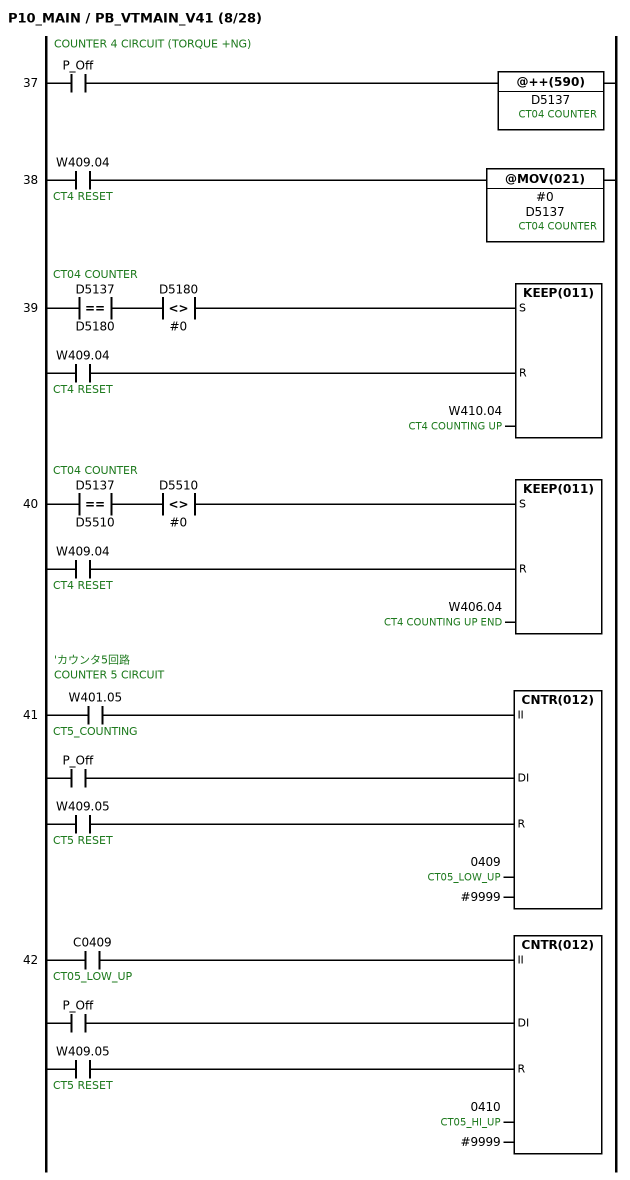
; rung 37: COUNTER 4 CIRCUIT (TORQUE +NG)
LD P_Off
@++(590) D5137  ; CT04 COUNTER
; rung 38
LD W409.04  ; CT4 RESET
@MOV(021) #0 D5137  ; CT04 COUNTER
; rung 39
LD=L(301) D5137 D5180  ; CT04 COUNTER
AND<>L(306) D5180 #0
LD W409.04  ; CT4 RESET
KEEP(011) W410.04  ; CT4 COUNTING UP
; rung 40
LD=L(301) D5137 D5510  ; CT04 COUNTER
AND<>L(306) D5510 #0
LD W409.04  ; CT4 RESET
KEEP(011) W406.04  ; CT4 COUNTING UP END
; rung 41: 'カウンタ5回路 / COUNTER 5 CIRCUIT
LD W401.05  ; CT5_COUNTING
LD P_Off
LD W409.05  ; CT5 RESET
CNTR(012) 0409 #9999  ; CT05_LOW_UP
; rung 42
LD C0409  ; CT05_LOW_UP
LD P_Off
LD W409.05  ; CT5 RESET
CNTR(012) 0410 #9999  ; CT05_HI_UP

